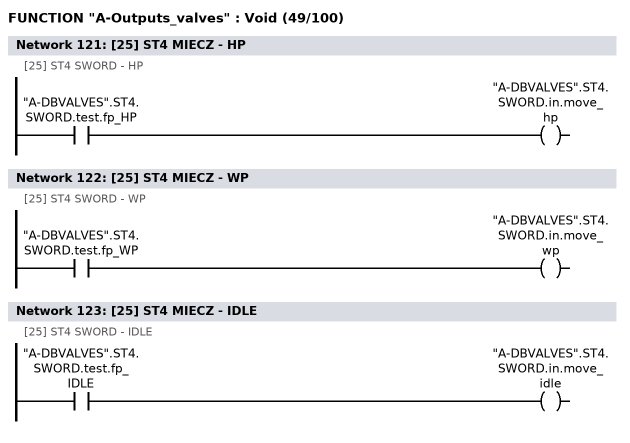
      O "A-DBVALVES".ST4.SWORD.test.fp_HP;
//    O     "A-Flags".STATION.IN_HP_STEP
      = "A-DBVALVES".ST4.SWORD.in.move_hp;
NETWORK
TITLE = [25] ST4 MIECZ - WP
//[25] ST4 SWORD - WP
      O "A-DBVALVES".ST4.SWORD.test.fp_WP;
      = "A-DBVALVES".ST4.SWORD.in.move_wp;
NETWORK
TITLE = [25] ST4 MIECZ - IDLE
//[25] ST4 SWORD - IDLE
      O "A-DBVALVES".ST4.SWORD.test.fp_IDLE;
      = "A-DBVALVES".ST4.SWORD.in.move_idle;
NETWORK
TITLE = [25] ST4 MIECZ
//[25] ST4 SWORD
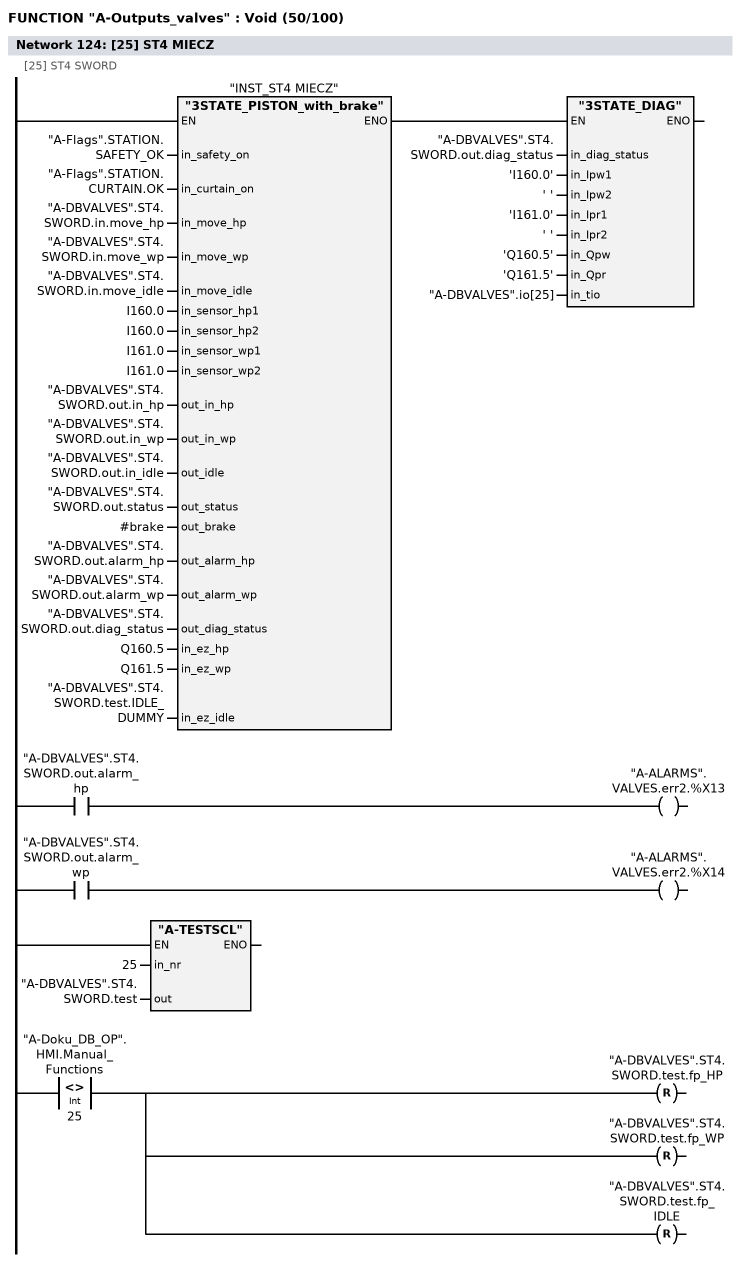
      CALL "3STATE_PISTON_with_brake", "INST_ST4 MIECZ"
      (  in_safety_on                := "A-Flags".STATION.SAFETY_OK ,
         in_curtain_on               := "A-Flags".STATION.CURTAIN.OK ,
         in_move_hp                  := "A-DBVALVES".ST4.SWORD.in.move_hp ,
         in_move_wp                  := "A-DBVALVES".ST4.SWORD.in.move_wp ,
         in_move_idle                := "A-DBVALVES".ST4.SWORD.in.move_idle ,
         in_sensor_hp1               := I160.0 ,
         in_sensor_hp2               := I160.0 ,
         in_sensor_wp1               := I161.0 ,
         in_sensor_wp2               := I161.0 ,
         out_in_hp                   := "A-DBVALVES".ST4.SWORD.out.in_hp ,
         out_in_wp                   := "A-DBVALVES".ST4.SWORD.out.in_wp ,
         out_idle                    := "A-DBVALVES".ST4.SWORD.out.in_idle ,
         out_status                  := "A-DBVALVES".ST4.SWORD.out.status ,
         out_brake                   := #brake ,
         out_alarm_hp                := "A-DBVALVES".ST4.SWORD.out.alarm_hp ,
         out_alarm_wp                := "A-DBVALVES".ST4.SWORD.out.alarm_wp ,
         out_diag_status             := "A-DBVALVES".ST4.SWORD.out.diag_status ,
         in_ez_hp                    := Q160.5 ,
         in_ez_wp                    := Q161.5 ,
         in_ez_idle                  := "A-DBVALVES".ST4.SWORD.test.IDLE_DUMMY
      );

      CALL "3STATE_DIAG"
      (  in_diag_status              := "A-DBVALVES".ST4.SWORD.out.diag_status ,
         in_Ipw1                     := 'I160.0' ,
         in_Ipw2                     := ' ' ,
         in_Ipr1                     := 'I161.0' ,
         in_Ipr2                     := ' ' ,
         in_Qpw                      := 'Q160.5' ,
         in_Qpr                      := 'Q161.5' ,
         in_tio                      := "A-DBVALVES".io[25]
      );

      A "A-DBVALVES".ST4.SWORD.out.alarm_hp;
      = "A-ALARMS".VALVES.err2.%X13;

      A "A-DBVALVES".ST4.SWORD.out.alarm_wp;
      = "A-ALARMS".VALVES.err2.%X14;

      CALL "A-TESTSCL"
      (  in_nr                       := 25 ,
         out                         := "A-DBVALVES".ST4.SWORD.test
      );

      A(;
      L "A-Doku_DB_OP".HMI.Manual_Functions;
      L 25;
      <>I;
      );
      R "A-DBVALVES".ST4.SWORD.test.fp_HP;
      R "A-DBVALVES".ST4.SWORD.test.fp_WP;
      R "A-DBVALVES".ST4.SWORD.test.fp_IDLE;
NETWORK
TITLE = -

NETWORK
TITLE = [26] ST4 ZDERZAK - HP
//[26] ST4 BUMPER - HP
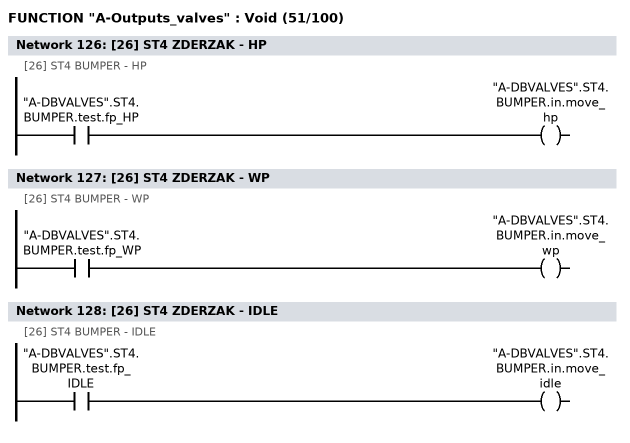
      O "A-DBVALVES".ST4.BUMPER.test.fp_HP;
//    O     "A-Flags".STATION.IN_HP_STEP
      = "A-DBVALVES".ST4.BUMPER.in.move_hp;
NETWORK
TITLE = [26] ST4 ZDERZAK - WP
//[26] ST4 BUMPER - WP
      O "A-DBVALVES".ST4.BUMPER.test.fp_WP;
      = "A-DBVALVES".ST4.BUMPER.in.move_wp;
NETWORK
TITLE = [26] ST4 ZDERZAK - IDLE
//[26] ST4 BUMPER - IDLE
      O "A-DBVALVES".ST4.BUMPER.test.fp_IDLE;
      = "A-DBVALVES".ST4.BUMPER.in.move_idle;
NETWORK
TITLE = [26] ST4 ZDERZAK
//[26] ST4 BUMPER
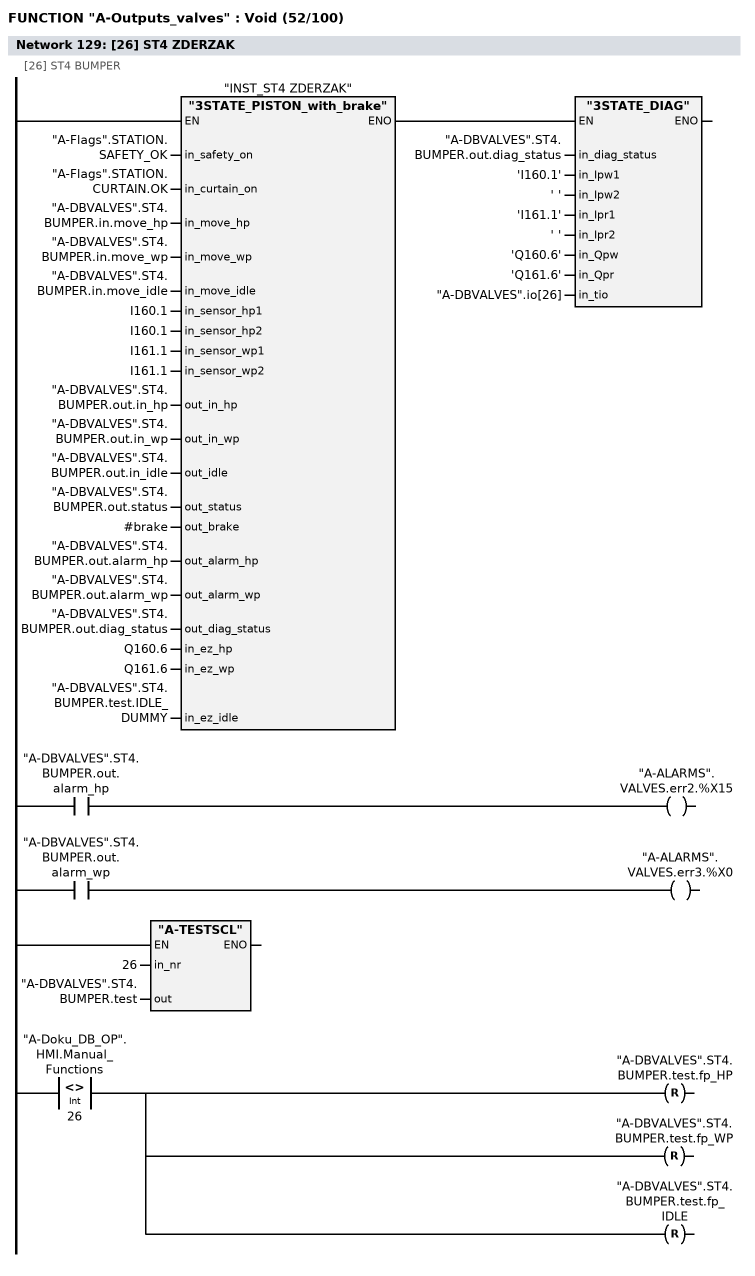
      CALL "3STATE_PISTON_with_brake", "INST_ST4 ZDERZAK"
      (  in_safety_on                := "A-Flags".STATION.SAFETY_OK ,
         in_curtain_on               := "A-Flags".STATION.CURTAIN.OK ,
         in_move_hp                  := "A-DBVALVES".ST4.BUMPER.in.move_hp ,
         in_move_wp                  := "A-DBVALVES".ST4.BUMPER.in.move_wp ,
         in_move_idle                := "A-DBVALVES".ST4.BUMPER.in.move_idle ,
         in_sensor_hp1               := I160.1 ,
         in_sensor_hp2               := I160.1 ,
         in_sensor_wp1               := I161.1 ,
         in_sensor_wp2               := I161.1 ,
         out_in_hp                   := "A-DBVALVES".ST4.BUMPER.out.in_hp ,
         out_in_wp                   := "A-DBVALVES".ST4.BUMPER.out.in_wp ,
         out_idle                    := "A-DBVALVES".ST4.BUMPER.out.in_idle ,
         out_status                  := "A-DBVALVES".ST4.BUMPER.out.status ,
         out_brake                   := #brake ,
         out_alarm_hp                := "A-DBVALVES".ST4.BUMPER.out.alarm_hp ,
         out_alarm_wp                := "A-DBVALVES".ST4.BUMPER.out.alarm_wp ,
         out_diag_status             := "A-DBVALVES".ST4.BUMPER.out.diag_status ,
         in_ez_hp                    := Q160.6 ,
         in_ez_wp                    := Q161.6 ,
         in_ez_idle                  := "A-DBVALVES".ST4.BUMPER.test.IDLE_DUMMY
      );

      CALL "3STATE_DIAG"
      (  in_diag_status              := "A-DBVALVES".ST4.BUMPER.out.diag_status ,
         in_Ipw1                     := 'I160.1' ,
         in_Ipw2                     := ' ' ,
         in_Ipr1                     := 'I161.1' ,
         in_Ipr2                     := ' ' ,
         in_Qpw                      := 'Q160.6' ,
         in_Qpr                      := 'Q161.6' ,
         in_tio                      := "A-DBVALVES".io[26]
      );

      A "A-DBVALVES".ST4.BUMPER.out.alarm_hp;
      = "A-ALARMS".VALVES.err2.%X15;

      A "A-DBVALVES".ST4.BUMPER.out.alarm_wp;
      = "A-ALARMS".VALVES.err3.%X0;

      CALL "A-TESTSCL"
      (  in_nr                       := 26 ,
         out                         := "A-DBVALVES".ST4.BUMPER.test
      );

      A(;
      L "A-Doku_DB_OP".HMI.Manual_Functions;
      L 26;
      <>I;
      );
      R "A-DBVALVES".ST4.BUMPER.test.fp_HP;
      R "A-DBVALVES".ST4.BUMPER.test.fp_WP;
      R "A-DBVALVES".ST4.BUMPER.test.fp_IDLE;
NETWORK
TITLE = -

NETWORK
TITLE = [27] ST4 PODNOSZENIE_MIECZA - HP
//[27] ST4 SWORD_RISING - HP
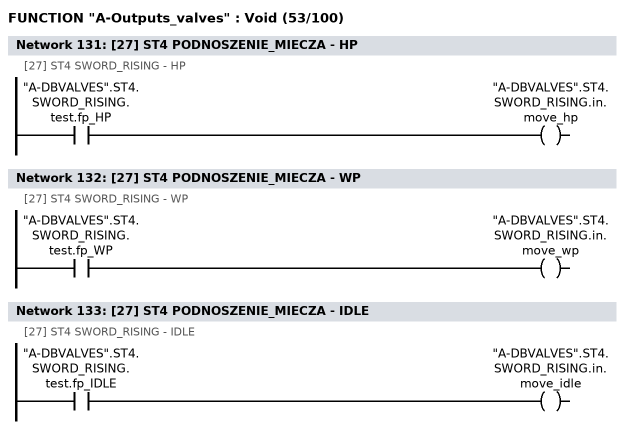
      O "A-DBVALVES".ST4.SWORD_RISING.test.fp_HP;
//    O     "A-Flags".STATION.IN_HP_STEP
      = "A-DBVALVES".ST4.SWORD_RISING.in.move_hp;
NETWORK
TITLE = [27] ST4 PODNOSZENIE_MIECZA - WP
//[27] ST4 SWORD_RISING - WP
      O "A-DBVALVES".ST4.SWORD_RISING.test.fp_WP;
      = "A-DBVALVES".ST4.SWORD_RISING.in.move_wp;
NETWORK
TITLE = [27] ST4 PODNOSZENIE_MIECZA - IDLE
//[27] ST4 SWORD_RISING - IDLE
      O "A-DBVALVES".ST4.SWORD_RISING.test.fp_IDLE;
      = "A-DBVALVES".ST4.SWORD_RISING.in.move_idle;
NETWORK
TITLE = [27] ST4 PODNOSZENIE_MIECZA
//[27] ST4 SWORD_RISING
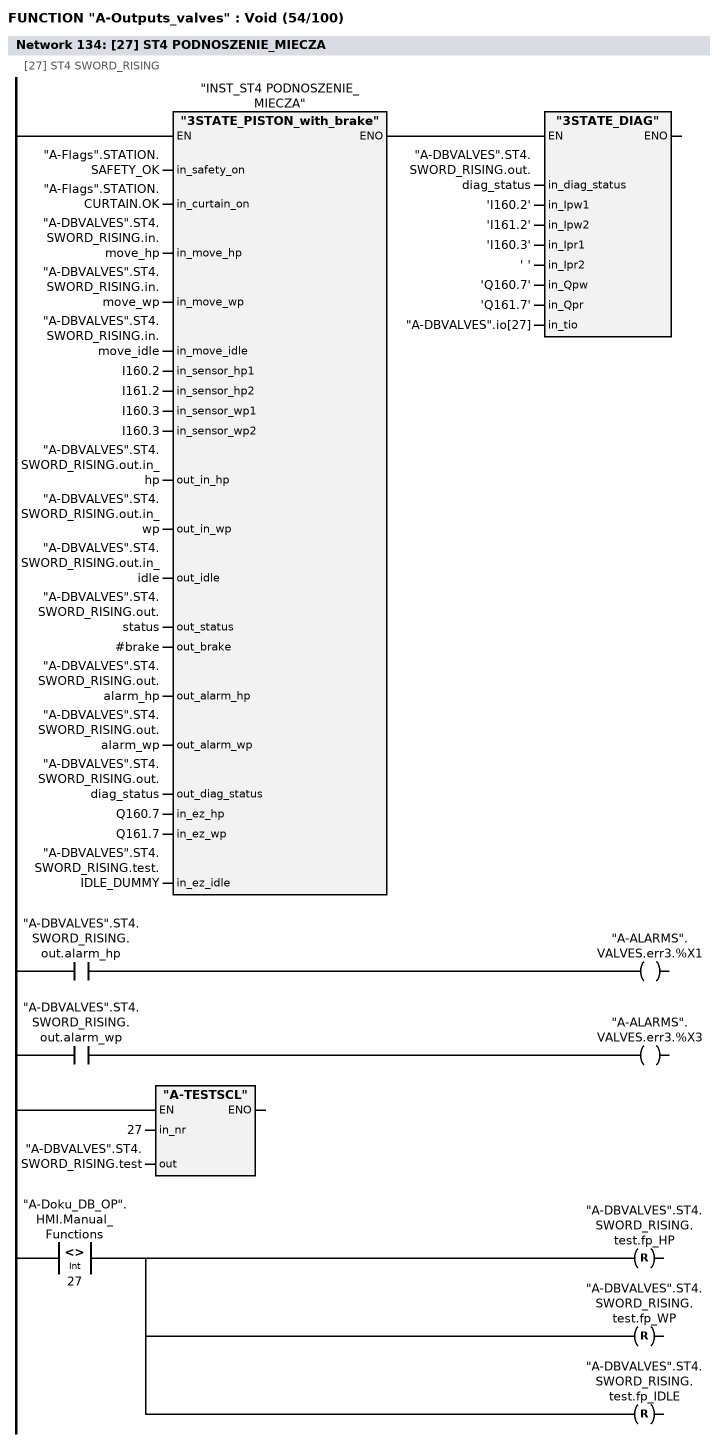
      CALL "3STATE_PISTON_with_brake", "INST_ST4 PODNOSZENIE_MIECZA"
      (  in_safety_on                := "A-Flags".STATION.SAFETY_OK ,
         in_curtain_on               := "A-Flags".STATION.CURTAIN.OK ,
         in_move_hp                  := "A-DBVALVES".ST4.SWORD_RISING.in.move_hp ,
         in_move_wp                  := "A-DBVALVES".ST4.SWORD_RISING.in.move_wp ,
         in_move_idle                := "A-DBVALVES".ST4.SWORD_RISING.in.move_idle ,
         in_sensor_hp1               := I160.2 ,
         in_sensor_hp2               := I161.2 ,
         in_sensor_wp1               := I160.3 ,
         in_sensor_wp2               := I160.3 ,
         out_in_hp                   := "A-DBVALVES".ST4.SWORD_RISING.out.in_hp ,
         out_in_wp                   := "A-DBVALVES".ST4.SWORD_RISING.out.in_wp ,
         out_idle                    := "A-DBVALVES".ST4.SWORD_RISING.out.in_idle ,
         out_status                  := "A-DBVALVES".ST4.SWORD_RISING.out.status ,
         out_brake                   := #brake ,
         out_alarm_hp                := "A-DBVALVES".ST4.SWORD_RISING.out.alarm_hp ,
         out_alarm_wp                := "A-DBVALVES".ST4.SWORD_RISING.out.alarm_wp ,
         out_diag_status             := "A-DBVALVES".ST4.SWORD_RISING.out.diag_status ,
         in_ez_hp                    := Q160.7 ,
         in_ez_wp                    := Q161.7 ,
         in_ez_idle                  := "A-DBVALVES".ST4.SWORD_RISING.test.IDLE_DUMMY
      );

      CALL "3STATE_DIAG"
      (  in_diag_status              := "A-DBVALVES".ST4.SWORD_RISING.out.diag_status ,
         in_Ipw1                     := 'I160.2' ,
         in_Ipw2                     := 'I161.2' ,
         in_Ipr1                     := 'I160.3' ,
         in_Ipr2                     := ' ' ,
         in_Qpw                      := 'Q160.7' ,
         in_Qpr                      := 'Q161.7' ,
         in_tio                      := "A-DBVALVES".io[27]
      );

      A "A-DBVALVES".ST4.SWORD_RISING.out.alarm_hp;
      = "A-ALARMS".VALVES.err3.%X1;

      A "A-DBVALVES".ST4.SWORD_RISING.out.alarm_wp;
      = "A-ALARMS".VALVES.err3.%X3;

      CALL "A-TESTSCL"
      (  in_nr                       := 27 ,
         out                         := "A-DBVALVES".ST4.SWORD_RISING.test
      );

      A(;
      L "A-Doku_DB_OP".HMI.Manual_Functions;
      L 27;
      <>I;
      );
      R "A-DBVALVES".ST4.SWORD_RISING.test.fp_HP;
      R "A-DBVALVES".ST4.SWORD_RISING.test.fp_WP;
      R "A-DBVALVES".ST4.SWORD_RISING.test.fp_IDLE;
NETWORK
TITLE = -

NETWORK
TITLE = [28] ST5 PRZESUW_STACJI - HP
//[28] ST5 STATION_MOVEMENT - HP
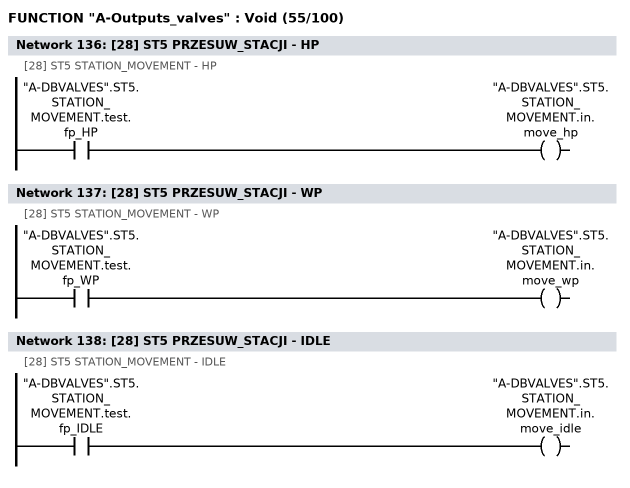
      O "A-DBVALVES".ST5.STATION_MOVEMENT.test.fp_HP;
//    O     "A-Flags".STATION.IN_HP_STEP
      = "A-DBVALVES".ST5.STATION_MOVEMENT.in.move_hp;
NETWORK
TITLE = [28] ST5 PRZESUW_STACJI - WP
//[28] ST5 STATION_MOVEMENT - WP
      O "A-DBVALVES".ST5.STATION_MOVEMENT.test.fp_WP;
      = "A-DBVALVES".ST5.STATION_MOVEMENT.in.move_wp;
NETWORK
TITLE = [28] ST5 PRZESUW_STACJI - IDLE
//[28] ST5 STATION_MOVEMENT - IDLE
      O "A-DBVALVES".ST5.STATION_MOVEMENT.test.fp_IDLE;
      = "A-DBVALVES".ST5.STATION_MOVEMENT.in.move_idle;
NETWORK
TITLE = [28] ST5 PRZESUW_STACJI
//[28] ST5 STATION_MOVEMENT
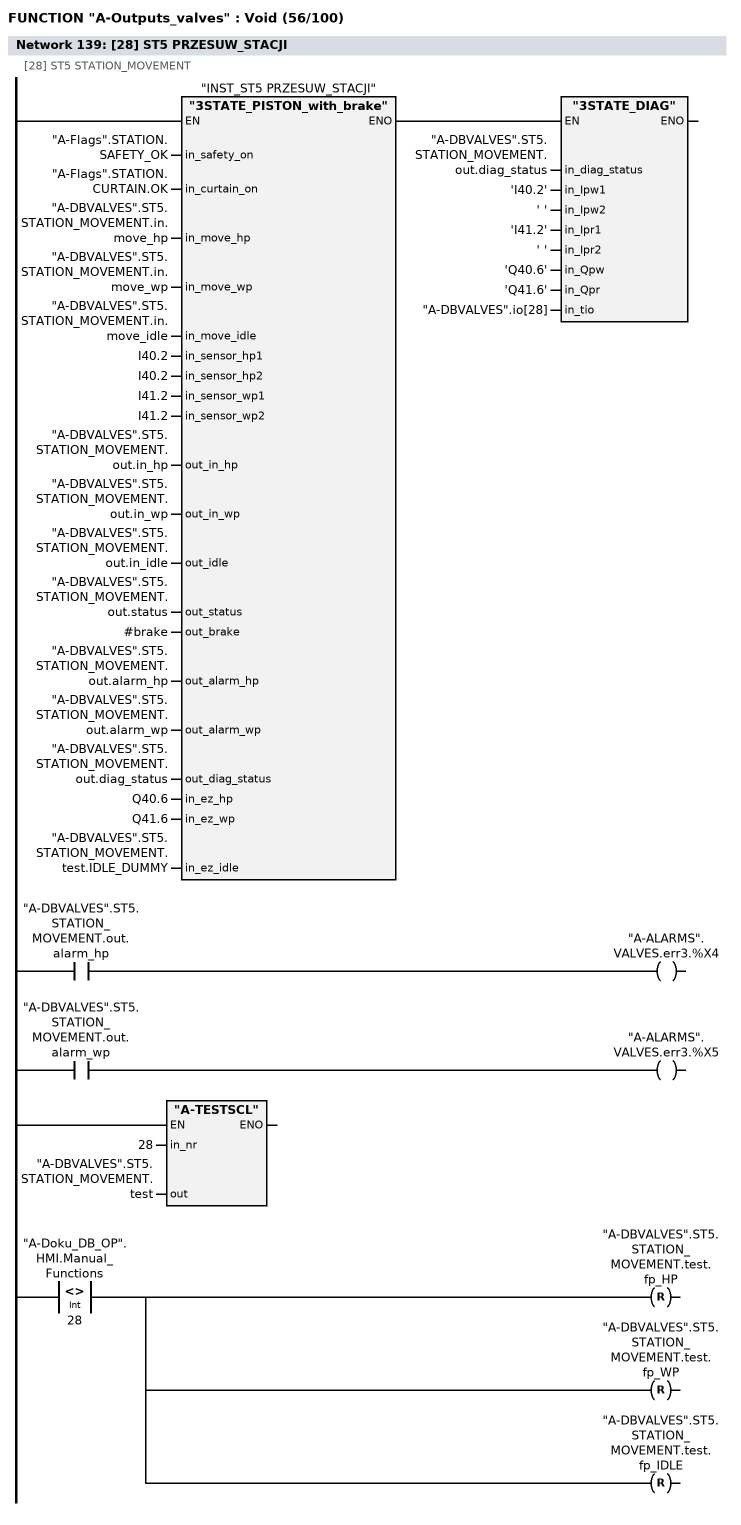
      CALL "3STATE_PISTON_with_brake", "INST_ST5 PRZESUW_STACJI"
      (  in_safety_on                := "A-Flags".STATION.SAFETY_OK ,
         in_curtain_on               := "A-Flags".STATION.CURTAIN.OK ,
         in_move_hp                  := "A-DBVALVES".ST5.STATION_MOVEMENT.in.move_hp ,
         in_move_wp                  := "A-DBVALVES".ST5.STATION_MOVEMENT.in.move_wp ,
         in_move_idle                := "A-DBVALVES".ST5.STATION_MOVEMENT.in.move_idle ,
         in_sensor_hp1               := I40.2 ,
         in_sensor_hp2               := I40.2 ,
         in_sensor_wp1               := I41.2 ,
         in_sensor_wp2               := I41.2 ,
         out_in_hp                   := "A-DBVALVES".ST5.STATION_MOVEMENT.out.in_hp ,
         out_in_wp                   := "A-DBVALVES".ST5.STATION_MOVEMENT.out.in_wp ,
         out_idle                    := "A-DBVALVES".ST5.STATION_MOVEMENT.out.in_idle ,
         out_status                  := "A-DBVALVES".ST5.STATION_MOVEMENT.out.status ,
         out_brake                   := #brake ,
         out_alarm_hp                := "A-DBVALVES".ST5.STATION_MOVEMENT.out.alarm_hp ,
         out_alarm_wp                := "A-DBVALVES".ST5.STATION_MOVEMENT.out.alarm_wp ,
         out_diag_status             := "A-DBVALVES".ST5.STATION_MOVEMENT.out.diag_status ,
         in_ez_hp                    := Q40.6 ,
         in_ez_wp                    := Q41.6 ,
         in_ez_idle                  := "A-DBVALVES".ST5.STATION_MOVEMENT.test.IDLE_DUMMY
      );

      CALL "3STATE_DIAG"
      (  in_diag_status              := "A-DBVALVES".ST5.STATION_MOVEMENT.out.diag_status ,
         in_Ipw1                     := 'I40.2' ,
         in_Ipw2                     := ' ' ,
         in_Ipr1                     := 'I41.2' ,
         in_Ipr2                     := ' ' ,
         in_Qpw                      := 'Q40.6' ,
         in_Qpr                      := 'Q41.6' ,
         in_tio                      := "A-DBVALVES".io[28]
      );

      A "A-DBVALVES".ST5.STATION_MOVEMENT.out.alarm_hp;
      = "A-ALARMS".VALVES.err3.%X4;

      A "A-DBVALVES".ST5.STATION_MOVEMENT.out.alarm_wp;
      = "A-ALARMS".VALVES.err3.%X5;

      CALL "A-TESTSCL"
      (  in_nr                       := 28 ,
         out                         := "A-DBVALVES".ST5.STATION_MOVEMENT.test
      );

      A(;
      L "A-Doku_DB_OP".HMI.Manual_Functions;
      L 28;
      <>I;
      );
      R "A-DBVALVES".ST5.STATION_MOVEMENT.test.fp_HP;
      R "A-DBVALVES".ST5.STATION_MOVEMENT.test.fp_WP;
      R "A-DBVALVES".ST5.STATION_MOVEMENT.test.fp_IDLE;
NETWORK
TITLE = -

NETWORK
TITLE = [29] ST5 STACJA_MALY_SKOK - HP
//[29] ST5 STATION_SMALL_STEP - HP
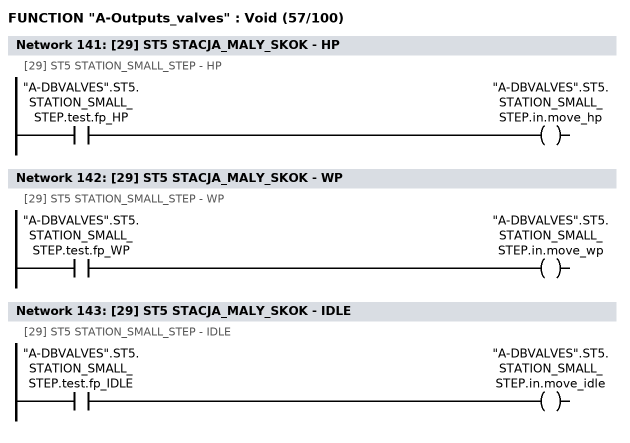
      O "A-DBVALVES".ST5.STATION_SMALL_STEP.test.fp_HP;
//    O     "A-Flags".STATION.IN_HP_STEP
      = "A-DBVALVES".ST5.STATION_SMALL_STEP.in.move_hp;
NETWORK
TITLE = [29] ST5 STACJA_MALY_SKOK - WP
//[29] ST5 STATION_SMALL_STEP - WP
      O "A-DBVALVES".ST5.STATION_SMALL_STEP.test.fp_WP;
      = "A-DBVALVES".ST5.STATION_SMALL_STEP.in.move_wp;
NETWORK
TITLE = [29] ST5 STACJA_MALY_SKOK - IDLE
//[29] ST5 STATION_SMALL_STEP - IDLE
      O "A-DBVALVES".ST5.STATION_SMALL_STEP.test.fp_IDLE;
      = "A-DBVALVES".ST5.STATION_SMALL_STEP.in.move_idle;
NETWORK
TITLE = [29] ST5 STACJA_MALY_SKOK
//[29] ST5 STATION_SMALL_STEP
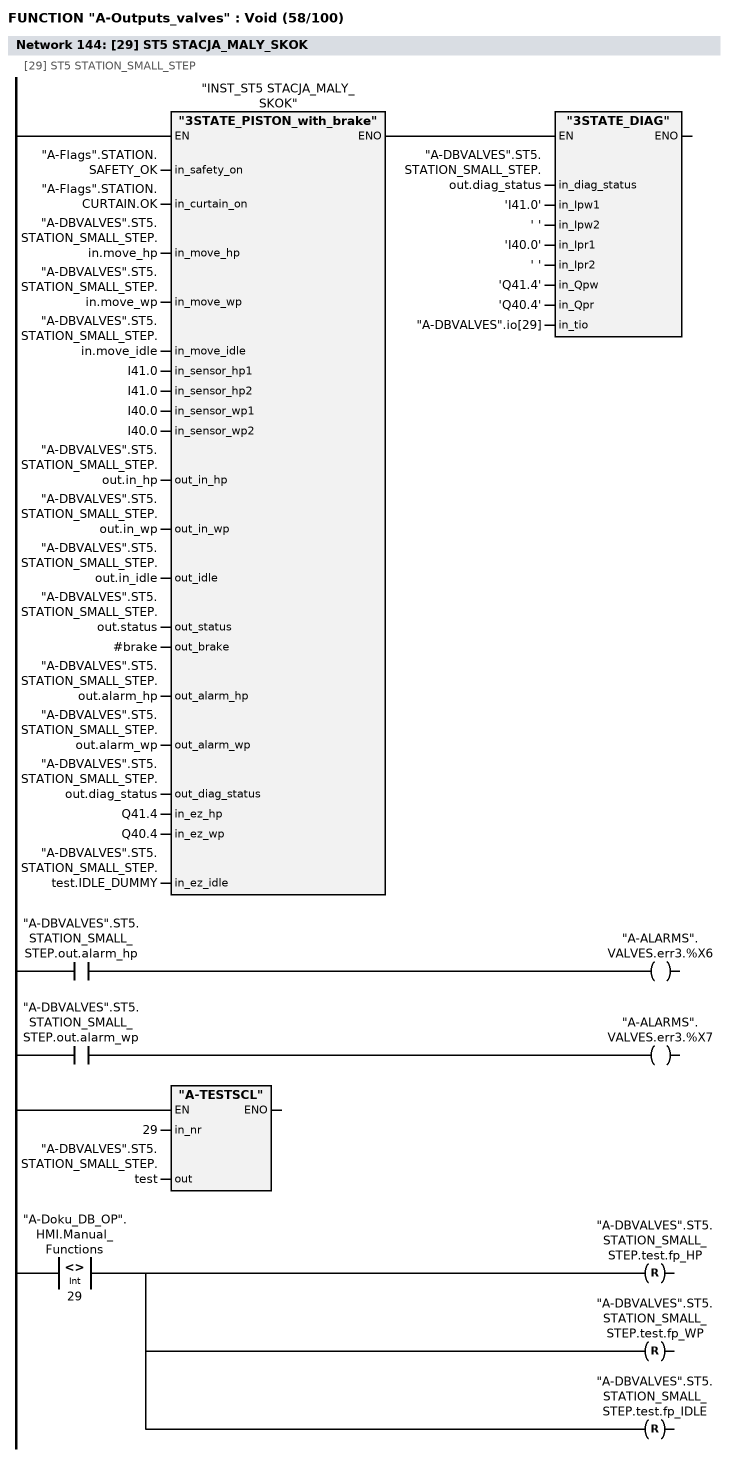
      CALL "3STATE_PISTON_with_brake", "INST_ST5 STACJA_MALY_SKOK"
      (  in_safety_on                := "A-Flags".STATION.SAFETY_OK ,
         in_curtain_on               := "A-Flags".STATION.CURTAIN.OK ,
         in_move_hp                  := "A-DBVALVES".ST5.STATION_SMALL_STEP.in.move_hp ,
         in_move_wp                  := "A-DBVALVES".ST5.STATION_SMALL_STEP.in.move_wp ,
         in_move_idle                := "A-DBVALVES".ST5.STATION_SMALL_STEP.in.move_idle ,
         in_sensor_hp1               := I41.0 ,
         in_sensor_hp2               := I41.0 ,
         in_sensor_wp1               := I40.0 ,
         in_sensor_wp2               := I40.0 ,
         out_in_hp                   := "A-DBVALVES".ST5.STATION_SMALL_STEP.out.in_hp ,
         out_in_wp                   := "A-DBVALVES".ST5.STATION_SMALL_STEP.out.in_wp ,
         out_idle                    := "A-DBVALVES".ST5.STATION_SMALL_STEP.out.in_idle ,
         out_status                  := "A-DBVALVES".ST5.STATION_SMALL_STEP.out.status ,
         out_brake                   := #brake ,
         out_alarm_hp                := "A-DBVALVES".ST5.STATION_SMALL_STEP.out.alarm_hp ,
         out_alarm_wp                := "A-DBVALVES".ST5.STATION_SMALL_STEP.out.alarm_wp ,
         out_diag_status             := "A-DBVALVES".ST5.STATION_SMALL_STEP.out.diag_status ,
         in_ez_hp                    := Q41.4 ,
         in_ez_wp                    := Q40.4 ,
         in_ez_idle                  := "A-DBVALVES".ST5.STATION_SMALL_STEP.test.IDLE_DUMMY
      );

      CALL "3STATE_DIAG"
      (  in_diag_status              := "A-DBVALVES".ST5.STATION_SMALL_STEP.out.diag_status ,
         in_Ipw1                     := 'I41.0' ,
         in_Ipw2                     := ' ' ,
         in_Ipr1                     := 'I40.0' ,
         in_Ipr2                     := ' ' ,
         in_Qpw                      := 'Q41.4' ,
         in_Qpr                      := 'Q40.4' ,
         in_tio                      := "A-DBVALVES".io[29]
      );

      A "A-DBVALVES".ST5.STATION_SMALL_STEP.out.alarm_hp;
      = "A-ALARMS".VALVES.err3.%X6;

      A "A-DBVALVES".ST5.STATION_SMALL_STEP.out.alarm_wp;
      = "A-ALARMS".VALVES.err3.%X7;

      CALL "A-TESTSCL"
      (  in_nr                       := 29 ,
         out                         := "A-DBVALVES".ST5.STATION_SMALL_STEP.test
      );

      A(;
      L "A-Doku_DB_OP".HMI.Manual_Functions;
      L 29;
      <>I;
      );
      R "A-DBVALVES".ST5.STATION_SMALL_STEP.test.fp_HP;
      R "A-DBVALVES".ST5.STATION_SMALL_STEP.test.fp_WP;
      R "A-DBVALVES".ST5.STATION_SMALL_STEP.test.fp_IDLE;
NETWORK
TITLE = -

NETWORK
TITLE = [30] ST5 STACJA_DUZY_SKOK - HP
//[30] ST5 STATION_BIG_STEP - HP
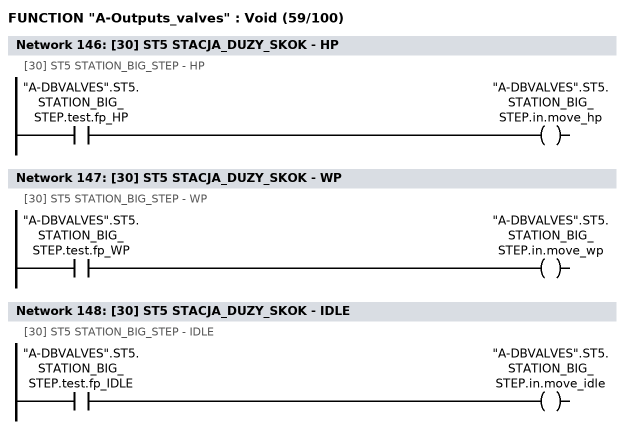
      O "A-DBVALVES".ST5.STATION_BIG_STEP.test.fp_HP;
//    O     "A-Flags".STATION.IN_HP_STEP
      = "A-DBVALVES".ST5.STATION_BIG_STEP.in.move_hp;
NETWORK
TITLE = [30] ST5 STACJA_DUZY_SKOK - WP
//[30] ST5 STATION_BIG_STEP - WP
      O "A-DBVALVES".ST5.STATION_BIG_STEP.test.fp_WP;
      = "A-DBVALVES".ST5.STATION_BIG_STEP.in.move_wp;
NETWORK
TITLE = [30] ST5 STACJA_DUZY_SKOK - IDLE
//[30] ST5 STATION_BIG_STEP - IDLE
      O "A-DBVALVES".ST5.STATION_BIG_STEP.test.fp_IDLE;
      = "A-DBVALVES".ST5.STATION_BIG_STEP.in.move_idle;
NETWORK
TITLE = [30] ST5 STACJA_DUZY_SKOK
//[30] ST5 STATION_BIG_STEP
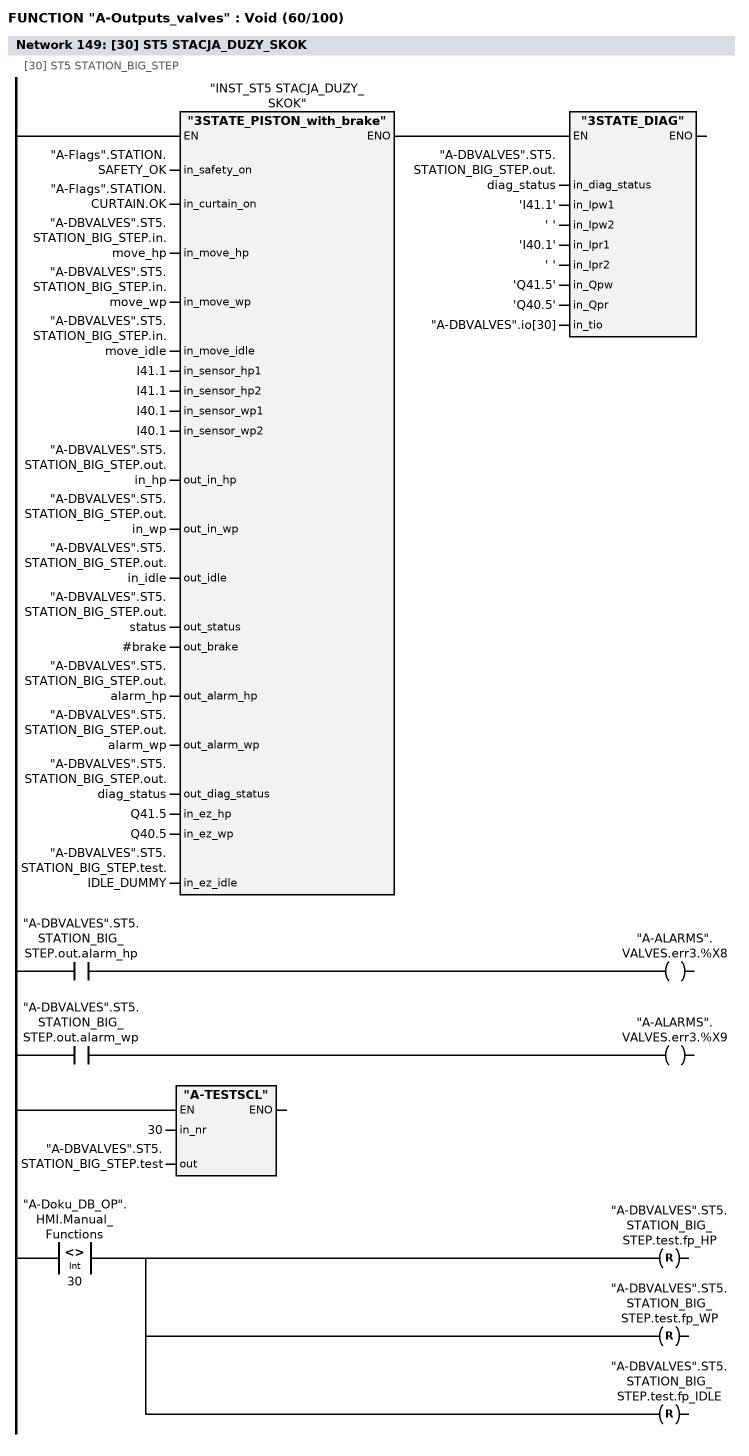
      CALL "3STATE_PISTON_with_brake", "INST_ST5 STACJA_DUZY_SKOK"
      (  in_safety_on                := "A-Flags".STATION.SAFETY_OK ,
         in_curtain_on               := "A-Flags".STATION.CURTAIN.OK ,
         in_move_hp                  := "A-DBVALVES".ST5.STATION_BIG_STEP.in.move_hp ,
         in_move_wp                  := "A-DBVALVES".ST5.STATION_BIG_STEP.in.move_wp ,
         in_move_idle                := "A-DBVALVES".ST5.STATION_BIG_STEP.in.move_idle ,
         in_sensor_hp1               := I41.1 ,
         in_sensor_hp2               := I41.1 ,
         in_sensor_wp1               := I40.1 ,
         in_sensor_wp2               := I40.1 ,
         out_in_hp                   := "A-DBVALVES".ST5.STATION_BIG_STEP.out.in_hp ,
         out_in_wp                   := "A-DBVALVES".ST5.STATION_BIG_STEP.out.in_wp ,
         out_idle                    := "A-DBVALVES".ST5.STATION_BIG_STEP.out.in_idle ,
         out_status                  := "A-DBVALVES".ST5.STATION_BIG_STEP.out.status ,
         out_brake                   := #brake ,
         out_alarm_hp                := "A-DBVALVES".ST5.STATION_BIG_STEP.out.alarm_hp ,
         out_alarm_wp                := "A-DBVALVES".ST5.STATION_BIG_STEP.out.alarm_wp ,
         out_diag_status             := "A-DBVALVES".ST5.STATION_BIG_STEP.out.diag_status ,
         in_ez_hp                    := Q41.5 ,
         in_ez_wp                    := Q40.5 ,
         in_ez_idle                  := "A-DBVALVES".ST5.STATION_BIG_STEP.test.IDLE_DUMMY
      );

      CALL "3STATE_DIAG"
      (  in_diag_status              := "A-DBVALVES".ST5.STATION_BIG_STEP.out.diag_status ,
         in_Ipw1                     := 'I41.1' ,
         in_Ipw2                     := ' ' ,
         in_Ipr1                     := 'I40.1' ,
         in_Ipr2                     := ' ' ,
         in_Qpw                      := 'Q41.5' ,
         in_Qpr                      := 'Q40.5' ,
         in_tio                      := "A-DBVALVES".io[30]
      );

      A "A-DBVALVES".ST5.STATION_BIG_STEP.out.alarm_hp;
      = "A-ALARMS".VALVES.err3.%X8;

      A "A-DBVALVES".ST5.STATION_BIG_STEP.out.alarm_wp;
      = "A-ALARMS".VALVES.err3.%X9;

      CALL "A-TESTSCL"
      (  in_nr                       := 30 ,
         out                         := "A-DBVALVES".ST5.STATION_BIG_STEP.test
      );

      A(;
      L "A-Doku_DB_OP".HMI.Manual_Functions;
      L 30;
      <>I;
      );
      R "A-DBVALVES".ST5.STATION_BIG_STEP.test.fp_HP;
      R "A-DBVALVES".ST5.STATION_BIG_STEP.test.fp_WP;
      R "A-DBVALVES".ST5.STATION_BIG_STEP.test.fp_IDLE;
NETWORK
TITLE = -

NETWORK
TITLE = [31] ST5 PIN - HP
//[31] ST5 PIN - HP
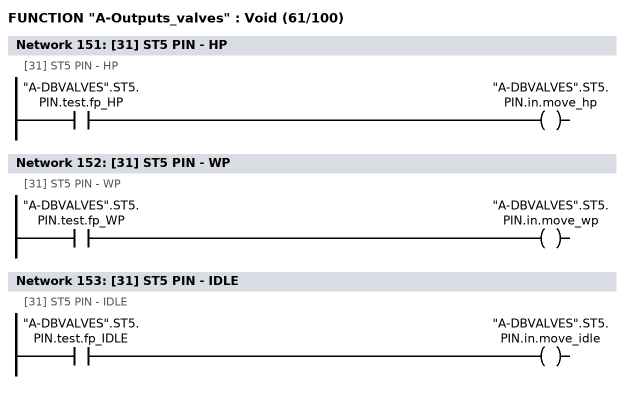
      O "A-DBVALVES".ST5.PIN.test.fp_HP;
//    O     "A-Flags".STATION.IN_HP_STEP
      = "A-DBVALVES".ST5.PIN.in.move_hp;
NETWORK
TITLE = [31] ST5 PIN - WP
//[31] ST5 PIN - WP
      O "A-DBVALVES".ST5.PIN.test.fp_WP;
      = "A-DBVALVES".ST5.PIN.in.move_wp;
NETWORK
TITLE = [31] ST5 PIN - IDLE
//[31] ST5 PIN - IDLE
      O "A-DBVALVES".ST5.PIN.test.fp_IDLE;
      = "A-DBVALVES".ST5.PIN.in.move_idle;
NETWORK
TITLE = [31] ST5 PIN
//[31] ST5 PIN
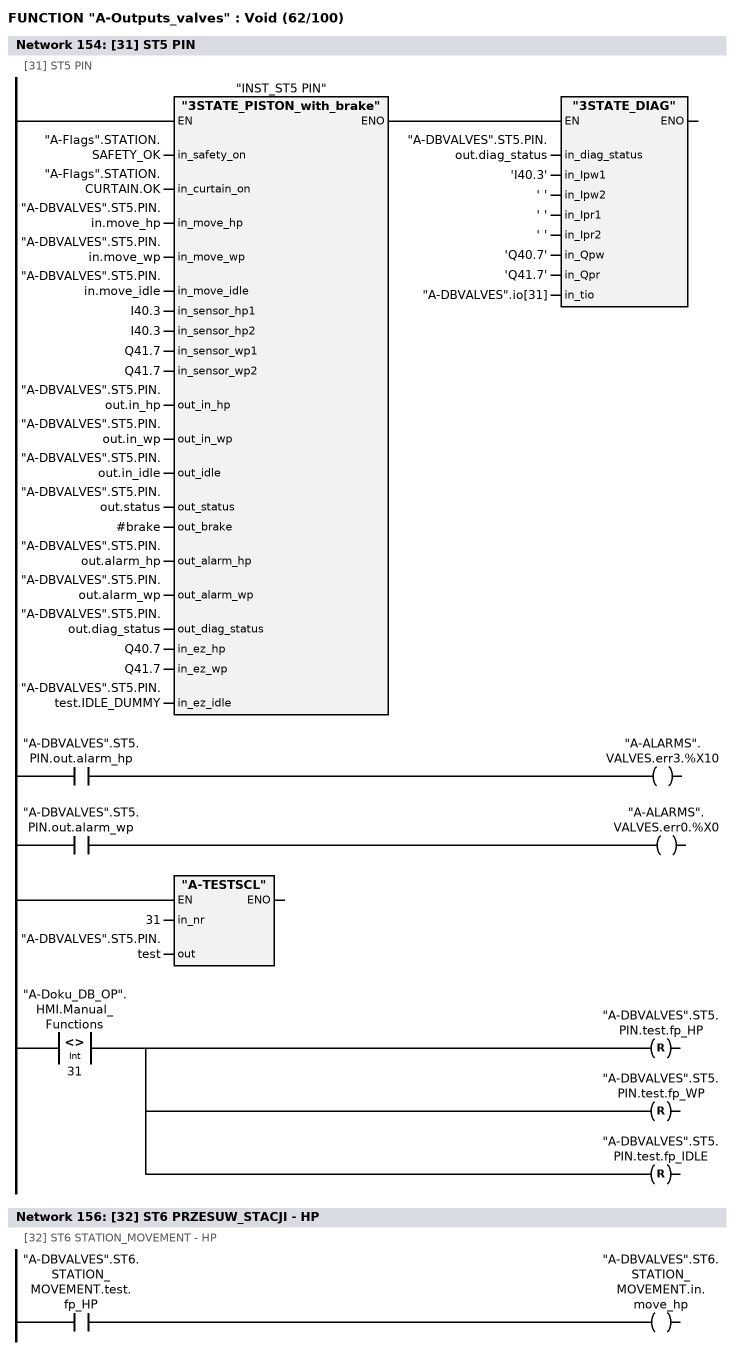
      CALL "3STATE_PISTON_with_brake", "INST_ST5 PIN"
      (  in_safety_on                := "A-Flags".STATION.SAFETY_OK ,
         in_curtain_on               := "A-Flags".STATION.CURTAIN.OK ,
         in_move_hp                  := "A-DBVALVES".ST5.PIN.in.move_hp ,
         in_move_wp                  := "A-DBVALVES".ST5.PIN.in.move_wp ,
         in_move_idle                := "A-DBVALVES".ST5.PIN.in.move_idle ,
         in_sensor_hp1               := I40.3 ,
         in_sensor_hp2               := I40.3 ,
         in_sensor_wp1               := Q41.7 ,
         in_sensor_wp2               := Q41.7 ,
         out_in_hp                   := "A-DBVALVES".ST5.PIN.out.in_hp ,
         out_in_wp                   := "A-DBVALVES".ST5.PIN.out.in_wp ,
         out_idle                    := "A-DBVALVES".ST5.PIN.out.in_idle ,
         out_status                  := "A-DBVALVES".ST5.PIN.out.status ,
         out_brake                   := #brake ,
         out_alarm_hp                := "A-DBVALVES".ST5.PIN.out.alarm_hp ,
         out_alarm_wp                := "A-DBVALVES".ST5.PIN.out.alarm_wp ,
         out_diag_status             := "A-DBVALVES".ST5.PIN.out.diag_status ,
         in_ez_hp                    := Q40.7 ,
         in_ez_wp                    := Q41.7 ,
         in_ez_idle                  := "A-DBVALVES".ST5.PIN.test.IDLE_DUMMY
      );

      CALL "3STATE_DIAG"
      (  in_diag_status              := "A-DBVALVES".ST5.PIN.out.diag_status ,
         in_Ipw1                     := 'I40.3' ,
         in_Ipw2                     := ' ' ,
         in_Ipr1                     := ' ' ,
         in_Ipr2                     := ' ' ,
         in_Qpw                      := 'Q40.7' ,
         in_Qpr                      := 'Q41.7' ,
         in_tio                      := "A-DBVALVES".io[31]
      );

      A "A-DBVALVES".ST5.PIN.out.alarm_hp;
      = "A-ALARMS".VALVES.err3.%X10;

      A "A-DBVALVES".ST5.PIN.out.alarm_wp;
      = "A-ALARMS".VALVES.err0.%X0;

      CALL "A-TESTSCL"
      (  in_nr                       := 31 ,
         out                         := "A-DBVALVES".ST5.PIN.test
      );

      A(;
      L "A-Doku_DB_OP".HMI.Manual_Functions;
      L 31;
      <>I;
      );
      R "A-DBVALVES".ST5.PIN.test.fp_HP;
      R "A-DBVALVES".ST5.PIN.test.fp_WP;
      R "A-DBVALVES".ST5.PIN.test.fp_IDLE;
NETWORK
TITLE = -

NETWORK
TITLE = [32] ST6 PRZESUW_STACJI - HP
//[32] ST6 STATION_MOVEMENT - HP
      O "A-DBVALVES".ST6.STATION_MOVEMENT.test.fp_HP;
//    O     "A-Flags".STATION.IN_HP_STEP
      = "A-DBVALVES".ST6.STATION_MOVEMENT.in.move_hp;
NETWORK
TITLE = [32] ST6 PRZESUW_STACJI - WP
//[32] ST6 STATION_MOVEMENT - WP
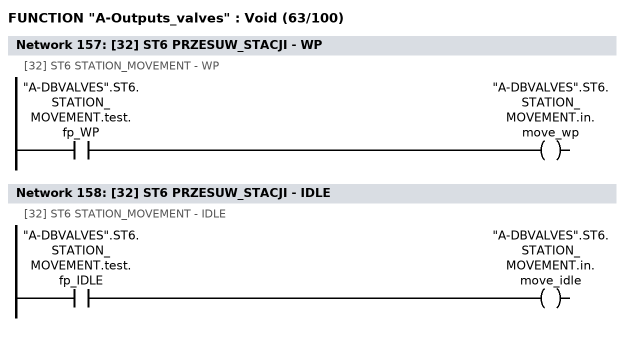
      O "A-DBVALVES".ST6.STATION_MOVEMENT.test.fp_WP;
      = "A-DBVALVES".ST6.STATION_MOVEMENT.in.move_wp;
NETWORK
TITLE = [32] ST6 PRZESUW_STACJI - IDLE
//[32] ST6 STATION_MOVEMENT - IDLE
      O "A-DBVALVES".ST6.STATION_MOVEMENT.test.fp_IDLE;
      = "A-DBVALVES".ST6.STATION_MOVEMENT.in.move_idle;
NETWORK
TITLE = [32] ST6 PRZESUW_STACJI
//[32] ST6 STATION_MOVEMENT
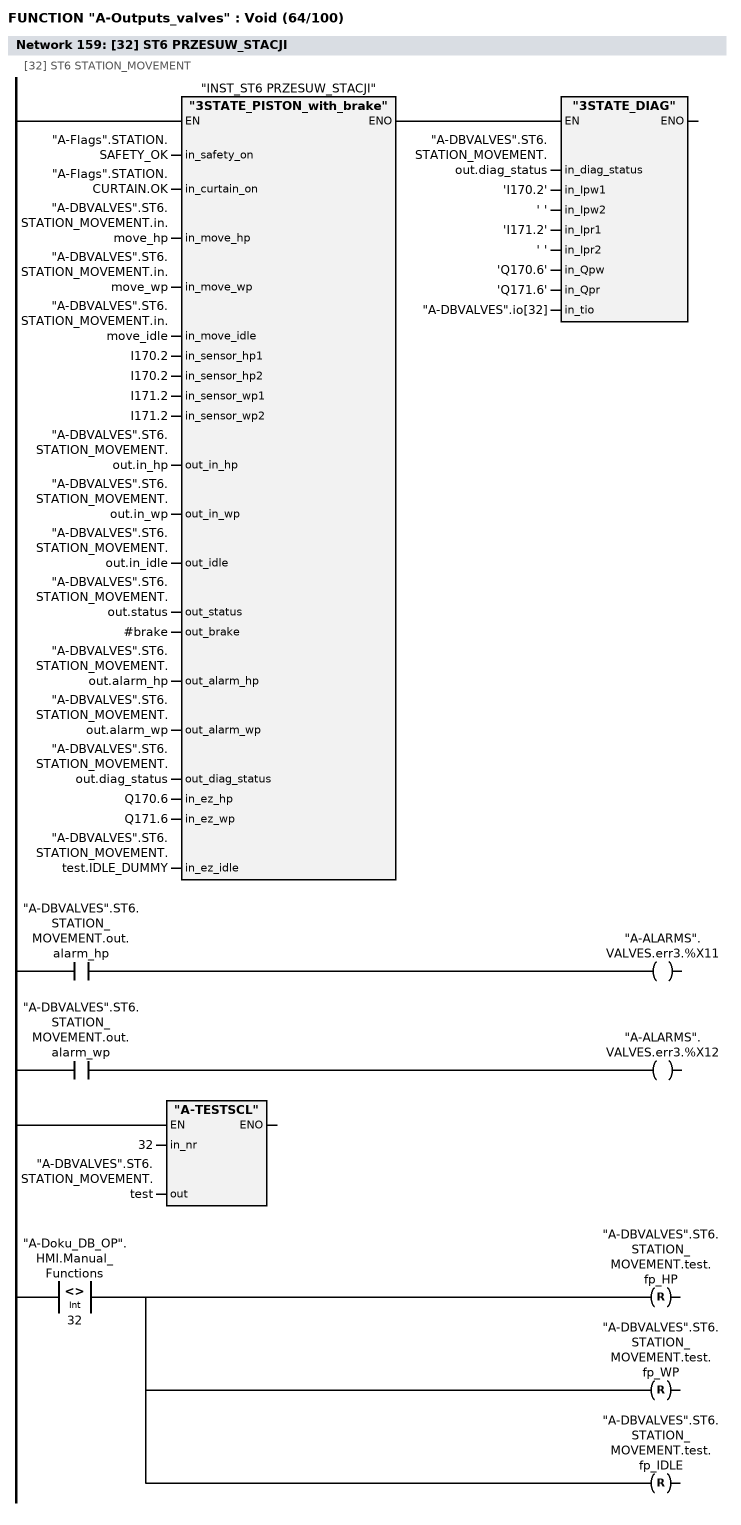
      CALL "3STATE_PISTON_with_brake", "INST_ST6 PRZESUW_STACJI"
      (  in_safety_on                := "A-Flags".STATION.SAFETY_OK ,
         in_curtain_on               := "A-Flags".STATION.CURTAIN.OK ,
         in_move_hp                  := "A-DBVALVES".ST6.STATION_MOVEMENT.in.move_hp ,
         in_move_wp                  := "A-DBVALVES".ST6.STATION_MOVEMENT.in.move_wp ,
         in_move_idle                := "A-DBVALVES".ST6.STATION_MOVEMENT.in.move_idle ,
         in_sensor_hp1               := I170.2 ,
         in_sensor_hp2               := I170.2 ,
         in_sensor_wp1               := I171.2 ,
         in_sensor_wp2               := I171.2 ,
         out_in_hp                   := "A-DBVALVES".ST6.STATION_MOVEMENT.out.in_hp ,
         out_in_wp                   := "A-DBVALVES".ST6.STATION_MOVEMENT.out.in_wp ,
         out_idle                    := "A-DBVALVES".ST6.STATION_MOVEMENT.out.in_idle ,
         out_status                  := "A-DBVALVES".ST6.STATION_MOVEMENT.out.status ,
         out_brake                   := #brake ,
         out_alarm_hp                := "A-DBVALVES".ST6.STATION_MOVEMENT.out.alarm_hp ,
         out_alarm_wp                := "A-DBVALVES".ST6.STATION_MOVEMENT.out.alarm_wp ,
         out_diag_status             := "A-DBVALVES".ST6.STATION_MOVEMENT.out.diag_status ,
         in_ez_hp                    := Q170.6 ,
         in_ez_wp                    := Q171.6 ,
         in_ez_idle                  := "A-DBVALVES".ST6.STATION_MOVEMENT.test.IDLE_DUMMY
      );

      CALL "3STATE_DIAG"
      (  in_diag_status              := "A-DBVALVES".ST6.STATION_MOVEMENT.out.diag_status ,
         in_Ipw1                     := 'I170.2' ,
         in_Ipw2                     := ' ' ,
         in_Ipr1                     := 'I171.2' ,
         in_Ipr2                     := ' ' ,
         in_Qpw                      := 'Q170.6' ,
         in_Qpr                      := 'Q171.6' ,
         in_tio                      := "A-DBVALVES".io[32]
      );

      A "A-DBVALVES".ST6.STATION_MOVEMENT.out.alarm_hp;
      = "A-ALARMS".VALVES.err3.%X11;

      A "A-DBVALVES".ST6.STATION_MOVEMENT.out.alarm_wp;
      = "A-ALARMS".VALVES.err3.%X12;

      CALL "A-TESTSCL"
      (  in_nr                       := 32 ,
         out                         := "A-DBVALVES".ST6.STATION_MOVEMENT.test
      );

      A(;
      L "A-Doku_DB_OP".HMI.Manual_Functions;
      L 32;
      <>I;
      );
      R "A-DBVALVES".ST6.STATION_MOVEMENT.test.fp_HP;
      R "A-DBVALVES".ST6.STATION_MOVEMENT.test.fp_WP;
      R "A-DBVALVES".ST6.STATION_MOVEMENT.test.fp_IDLE;
NETWORK
TITLE = -

NETWORK
TITLE = [33] ST6 STACJA_MALY_SKOK - HP
//[33] ST6 STATION_SMALL_STEP - HP
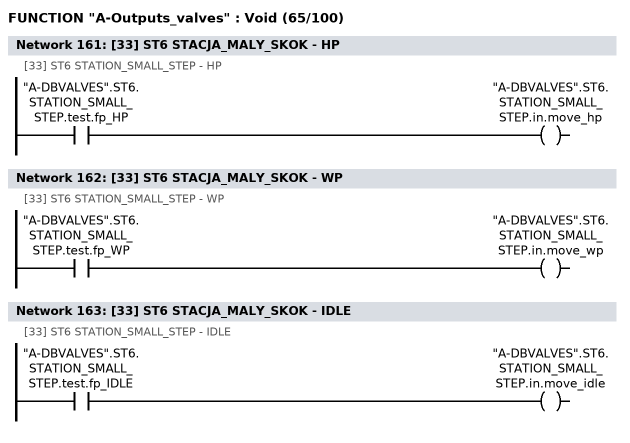
      O "A-DBVALVES".ST6.STATION_SMALL_STEP.test.fp_HP;
//    O     "A-Flags".STATION.IN_HP_STEP
      = "A-DBVALVES".ST6.STATION_SMALL_STEP.in.move_hp;
NETWORK
TITLE = [33] ST6 STACJA_MALY_SKOK - WP
//[33] ST6 STATION_SMALL_STEP - WP
      O "A-DBVALVES".ST6.STATION_SMALL_STEP.test.fp_WP;
      = "A-DBVALVES".ST6.STATION_SMALL_STEP.in.move_wp;
NETWORK
TITLE = [33] ST6 STACJA_MALY_SKOK - IDLE
//[33] ST6 STATION_SMALL_STEP - IDLE
      O "A-DBVALVES".ST6.STATION_SMALL_STEP.test.fp_IDLE;
      = "A-DBVALVES".ST6.STATION_SMALL_STEP.in.move_idle;
NETWORK
TITLE = [33] ST6 STACJA_MALY_SKOK
//[33] ST6 STATION_SMALL_STEP
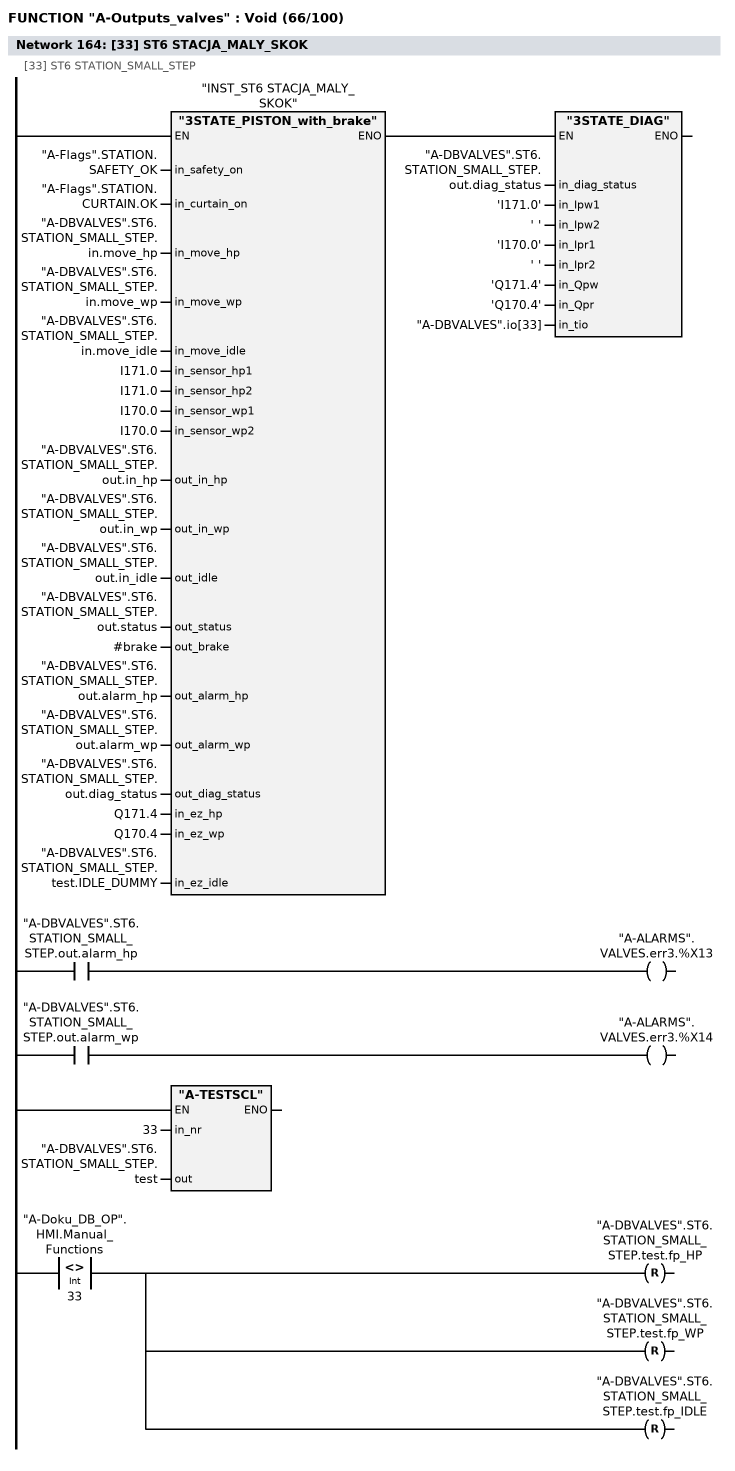
      CALL "3STATE_PISTON_with_brake", "INST_ST6 STACJA_MALY_SKOK"
      (  in_safety_on                := "A-Flags".STATION.SAFETY_OK ,
         in_curtain_on               := "A-Flags".STATION.CURTAIN.OK ,
         in_move_hp                  := "A-DBVALVES".ST6.STATION_SMALL_STEP.in.move_hp ,
         in_move_wp                  := "A-DBVALVES".ST6.STATION_SMALL_STEP.in.move_wp ,
         in_move_idle                := "A-DBVALVES".ST6.STATION_SMALL_STEP.in.move_idle ,
         in_sensor_hp1               := I171.0 ,
         in_sensor_hp2               := I171.0 ,
         in_sensor_wp1               := I170.0 ,
         in_sensor_wp2               := I170.0 ,
         out_in_hp                   := "A-DBVALVES".ST6.STATION_SMALL_STEP.out.in_hp ,
         out_in_wp                   := "A-DBVALVES".ST6.STATION_SMALL_STEP.out.in_wp ,
         out_idle                    := "A-DBVALVES".ST6.STATION_SMALL_STEP.out.in_idle ,
         out_status                  := "A-DBVALVES".ST6.STATION_SMALL_STEP.out.status ,
         out_brake                   := #brake ,
         out_alarm_hp                := "A-DBVALVES".ST6.STATION_SMALL_STEP.out.alarm_hp ,
         out_alarm_wp                := "A-DBVALVES".ST6.STATION_SMALL_STEP.out.alarm_wp ,
         out_diag_status             := "A-DBVALVES".ST6.STATION_SMALL_STEP.out.diag_status ,
         in_ez_hp                    := Q171.4 ,
         in_ez_wp                    := Q170.4 ,
         in_ez_idle                  := "A-DBVALVES".ST6.STATION_SMALL_STEP.test.IDLE_DUMMY
      );

      CALL "3STATE_DIAG"
      (  in_diag_status              := "A-DBVALVES".ST6.STATION_SMALL_STEP.out.diag_status ,
         in_Ipw1                     := 'I171.0' ,
         in_Ipw2                     := ' ' ,
         in_Ipr1                     := 'I170.0' ,
         in_Ipr2                     := ' ' ,
         in_Qpw                      := 'Q171.4' ,
         in_Qpr                      := 'Q170.4' ,
         in_tio                      := "A-DBVALVES".io[33]
      );

      A "A-DBVALVES".ST6.STATION_SMALL_STEP.out.alarm_hp;
      = "A-ALARMS".VALVES.err3.%X13;

      A "A-DBVALVES".ST6.STATION_SMALL_STEP.out.alarm_wp;
      = "A-ALARMS".VALVES.err3.%X14;

      CALL "A-TESTSCL"
      (  in_nr                       := 33 ,
         out                         := "A-DBVALVES".ST6.STATION_SMALL_STEP.test
      );

      A(;
      L "A-Doku_DB_OP".HMI.Manual_Functions;
      L 33;
      <>I;
      );
      R "A-DBVALVES".ST6.STATION_SMALL_STEP.test.fp_HP;
      R "A-DBVALVES".ST6.STATION_SMALL_STEP.test.fp_WP;
      R "A-DBVALVES".ST6.STATION_SMALL_STEP.test.fp_IDLE;
NETWORK
TITLE = -

NETWORK
TITLE = [34] ST6 STACJA_DUZY_SKOK - HP
//[34] ST6 STATION_BIG_STEP - HP
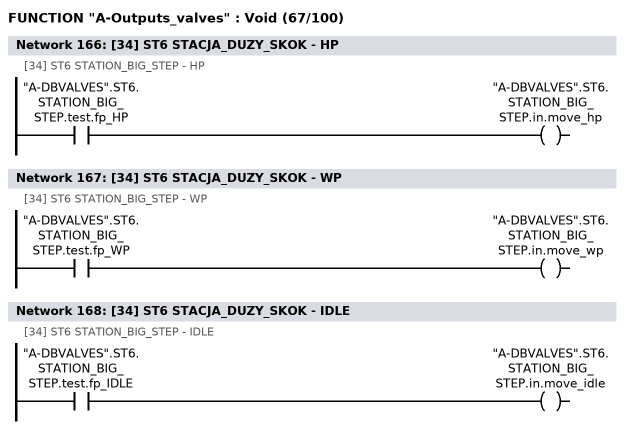
      O "A-DBVALVES".ST6.STATION_BIG_STEP.test.fp_HP;
//    O     "A-Flags".STATION.IN_HP_STEP
      = "A-DBVALVES".ST6.STATION_BIG_STEP.in.move_hp;
NETWORK
TITLE = [34] ST6 STACJA_DUZY_SKOK - WP
//[34] ST6 STATION_BIG_STEP - WP
      O "A-DBVALVES".ST6.STATION_BIG_STEP.test.fp_WP;
      = "A-DBVALVES".ST6.STATION_BIG_STEP.in.move_wp;
NETWORK
TITLE = [34] ST6 STACJA_DUZY_SKOK - IDLE
//[34] ST6 STATION_BIG_STEP - IDLE
      O "A-DBVALVES".ST6.STATION_BIG_STEP.test.fp_IDLE;
      = "A-DBVALVES".ST6.STATION_BIG_STEP.in.move_idle;
NETWORK
TITLE = [34] ST6 STACJA_DUZY_SKOK
//[34] ST6 STATION_BIG_STEP
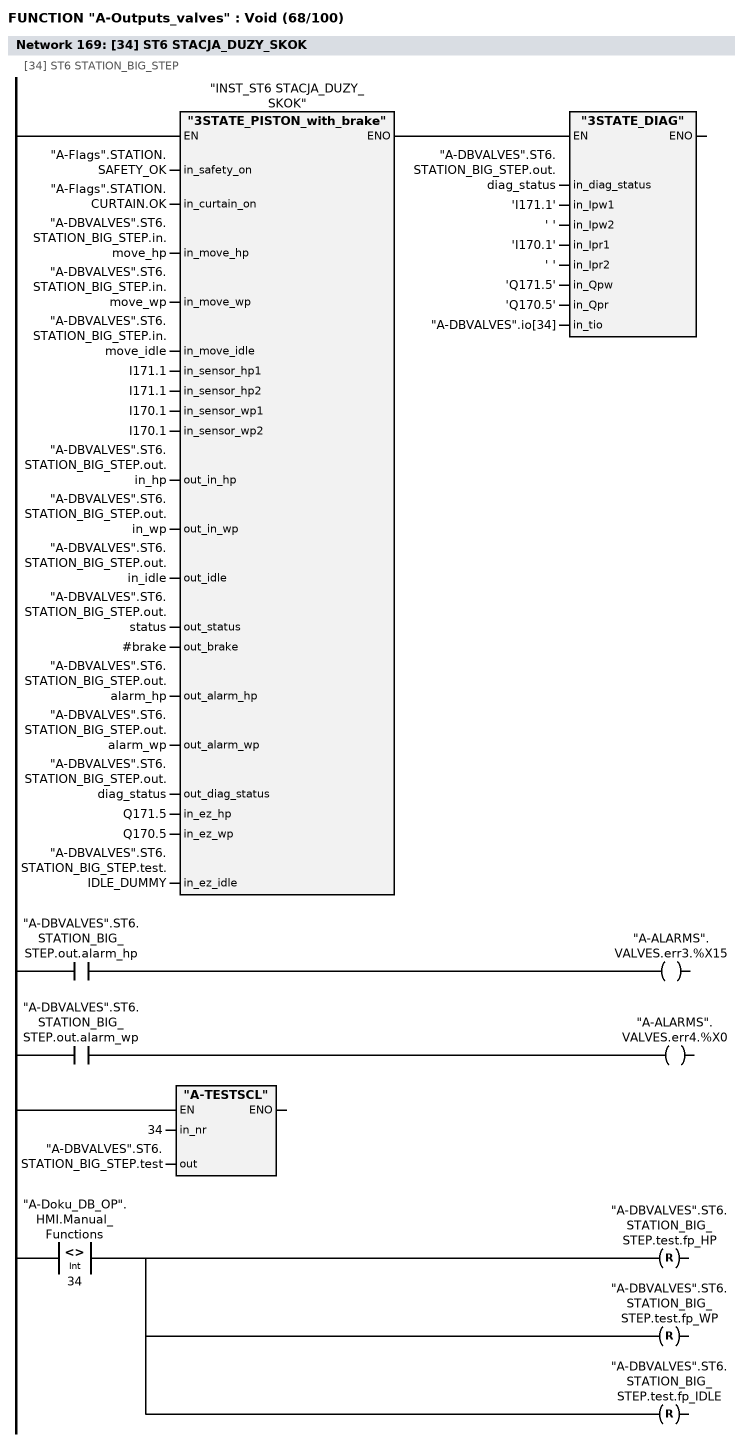
      CALL "3STATE_PISTON_with_brake", "INST_ST6 STACJA_DUZY_SKOK"
      (  in_safety_on                := "A-Flags".STATION.SAFETY_OK ,
         in_curtain_on               := "A-Flags".STATION.CURTAIN.OK ,
         in_move_hp                  := "A-DBVALVES".ST6.STATION_BIG_STEP.in.move_hp ,
         in_move_wp                  := "A-DBVALVES".ST6.STATION_BIG_STEP.in.move_wp ,
         in_move_idle                := "A-DBVALVES".ST6.STATION_BIG_STEP.in.move_idle ,
         in_sensor_hp1               := I171.1 ,
         in_sensor_hp2               := I171.1 ,
         in_sensor_wp1               := I170.1 ,
         in_sensor_wp2               := I170.1 ,
         out_in_hp                   := "A-DBVALVES".ST6.STATION_BIG_STEP.out.in_hp ,
         out_in_wp                   := "A-DBVALVES".ST6.STATION_BIG_STEP.out.in_wp ,
         out_idle                    := "A-DBVALVES".ST6.STATION_BIG_STEP.out.in_idle ,
         out_status                  := "A-DBVALVES".ST6.STATION_BIG_STEP.out.status ,
         out_brake                   := #brake ,
         out_alarm_hp                := "A-DBVALVES".ST6.STATION_BIG_STEP.out.alarm_hp ,
         out_alarm_wp                := "A-DBVALVES".ST6.STATION_BIG_STEP.out.alarm_wp ,
         out_diag_status             := "A-DBVALVES".ST6.STATION_BIG_STEP.out.diag_status ,
         in_ez_hp                    := Q171.5 ,
         in_ez_wp                    := Q170.5 ,
         in_ez_idle                  := "A-DBVALVES".ST6.STATION_BIG_STEP.test.IDLE_DUMMY
      );

      CALL "3STATE_DIAG"
      (  in_diag_status              := "A-DBVALVES".ST6.STATION_BIG_STEP.out.diag_status ,
         in_Ipw1                     := 'I171.1' ,
         in_Ipw2                     := ' ' ,
         in_Ipr1                     := 'I170.1' ,
         in_Ipr2                     := ' ' ,
         in_Qpw                      := 'Q171.5' ,
         in_Qpr                      := 'Q170.5' ,
         in_tio                      := "A-DBVALVES".io[34]
      );

      A "A-DBVALVES".ST6.STATION_BIG_STEP.out.alarm_hp;
      = "A-ALARMS".VALVES.err3.%X15;

      A "A-DBVALVES".ST6.STATION_BIG_STEP.out.alarm_wp;
      = "A-ALARMS".VALVES.err4.%X0;

      CALL "A-TESTSCL"
      (  in_nr                       := 34 ,
         out                         := "A-DBVALVES".ST6.STATION_BIG_STEP.test
      );

      A(;
      L "A-Doku_DB_OP".HMI.Manual_Functions;
      L 34;
      <>I;
      );
      R "A-DBVALVES".ST6.STATION_BIG_STEP.test.fp_HP;
      R "A-DBVALVES".ST6.STATION_BIG_STEP.test.fp_WP;
      R "A-DBVALVES".ST6.STATION_BIG_STEP.test.fp_IDLE;
NETWORK
TITLE = -

NETWORK
TITLE = [35] ST6 PIN - HP
//[35] ST6 PIN - HP
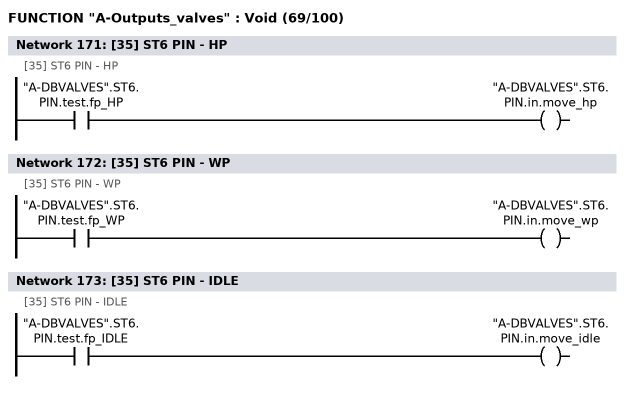
      O "A-DBVALVES".ST6.PIN.test.fp_HP;
//    O     "A-Flags".STATION.IN_HP_STEP
      = "A-DBVALVES".ST6.PIN.in.move_hp;
NETWORK
TITLE = [35] ST6 PIN - WP
//[35] ST6 PIN - WP
      O "A-DBVALVES".ST6.PIN.test.fp_WP;
      = "A-DBVALVES".ST6.PIN.in.move_wp;
NETWORK
TITLE = [35] ST6 PIN - IDLE
//[35] ST6 PIN - IDLE
      O "A-DBVALVES".ST6.PIN.test.fp_IDLE;
      = "A-DBVALVES".ST6.PIN.in.move_idle;
NETWORK
TITLE = [35] ST6 PIN
//[35] ST6 PIN
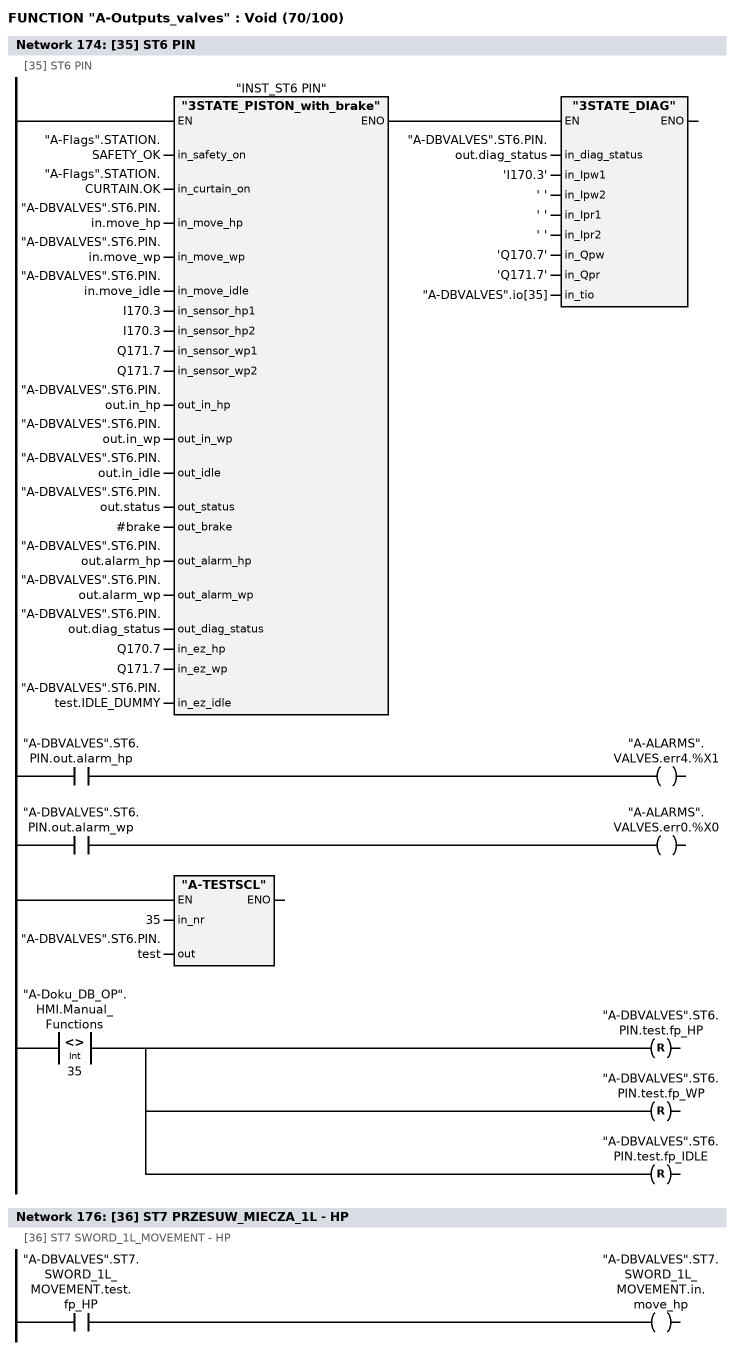
      CALL "3STATE_PISTON_with_brake", "INST_ST6 PIN"
      (  in_safety_on                := "A-Flags".STATION.SAFETY_OK ,
         in_curtain_on               := "A-Flags".STATION.CURTAIN.OK ,
         in_move_hp                  := "A-DBVALVES".ST6.PIN.in.move_hp ,
         in_move_wp                  := "A-DBVALVES".ST6.PIN.in.move_wp ,
         in_move_idle                := "A-DBVALVES".ST6.PIN.in.move_idle ,
         in_sensor_hp1               := I170.3 ,
         in_sensor_hp2               := I170.3 ,
         in_sensor_wp1               := Q171.7 ,
         in_sensor_wp2               := Q171.7 ,
         out_in_hp                   := "A-DBVALVES".ST6.PIN.out.in_hp ,
         out_in_wp                   := "A-DBVALVES".ST6.PIN.out.in_wp ,
         out_idle                    := "A-DBVALVES".ST6.PIN.out.in_idle ,
         out_status                  := "A-DBVALVES".ST6.PIN.out.status ,
         out_brake                   := #brake ,
         out_alarm_hp                := "A-DBVALVES".ST6.PIN.out.alarm_hp ,
         out_alarm_wp                := "A-DBVALVES".ST6.PIN.out.alarm_wp ,
         out_diag_status             := "A-DBVALVES".ST6.PIN.out.diag_status ,
         in_ez_hp                    := Q170.7 ,
         in_ez_wp                    := Q171.7 ,
         in_ez_idle                  := "A-DBVALVES".ST6.PIN.test.IDLE_DUMMY
      );

      CALL "3STATE_DIAG"
      (  in_diag_status              := "A-DBVALVES".ST6.PIN.out.diag_status ,
         in_Ipw1                     := 'I170.3' ,
         in_Ipw2                     := ' ' ,
         in_Ipr1                     := ' ' ,
         in_Ipr2                     := ' ' ,
         in_Qpw                      := 'Q170.7' ,
         in_Qpr                      := 'Q171.7' ,
         in_tio                      := "A-DBVALVES".io[35]
      );

      A "A-DBVALVES".ST6.PIN.out.alarm_hp;
      = "A-ALARMS".VALVES.err4.%X1;

      A "A-DBVALVES".ST6.PIN.out.alarm_wp;
      = "A-ALARMS".VALVES.err0.%X0;

      CALL "A-TESTSCL"
      (  in_nr                       := 35 ,
         out                         := "A-DBVALVES".ST6.PIN.test
      );

      A(;
      L "A-Doku_DB_OP".HMI.Manual_Functions;
      L 35;
      <>I;
      );
      R "A-DBVALVES".ST6.PIN.test.fp_HP;
      R "A-DBVALVES".ST6.PIN.test.fp_WP;
      R "A-DBVALVES".ST6.PIN.test.fp_IDLE;
NETWORK
TITLE = -

NETWORK
TITLE = [36] ST7 PRZESUW_MIECZA_1L - HP
//[36] ST7 SWORD_1L_MOVEMENT - HP
      O "A-DBVALVES".ST7.SWORD_1L_MOVEMENT.test.fp_HP;
//    O     "A-Flags".STATION.IN_HP_STEP
      = "A-DBVALVES".ST7.SWORD_1L_MOVEMENT.in.move_hp;
NETWORK
TITLE = [36] ST7 PRZESUW_MIECZA_1L - WP
//[36] ST7 SWORD_1L_MOVEMENT - WP
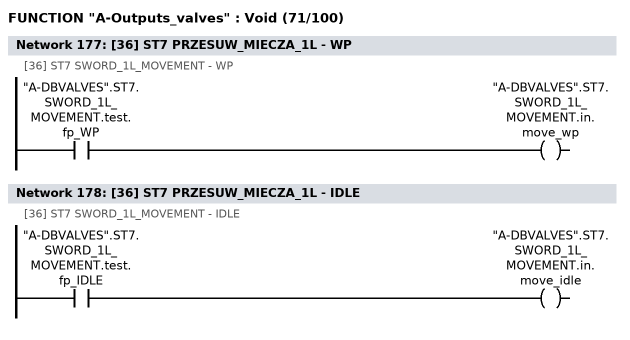
      O "A-DBVALVES".ST7.SWORD_1L_MOVEMENT.test.fp_WP;
      = "A-DBVALVES".ST7.SWORD_1L_MOVEMENT.in.move_wp;
NETWORK
TITLE = [36] ST7 PRZESUW_MIECZA_1L - IDLE
//[36] ST7 SWORD_1L_MOVEMENT - IDLE
      O "A-DBVALVES".ST7.SWORD_1L_MOVEMENT.test.fp_IDLE;
      = "A-DBVALVES".ST7.SWORD_1L_MOVEMENT.in.move_idle;
NETWORK
TITLE = [36] ST7 PRZESUW_MIECZA_1L
//[36] ST7 SWORD_1L_MOVEMENT
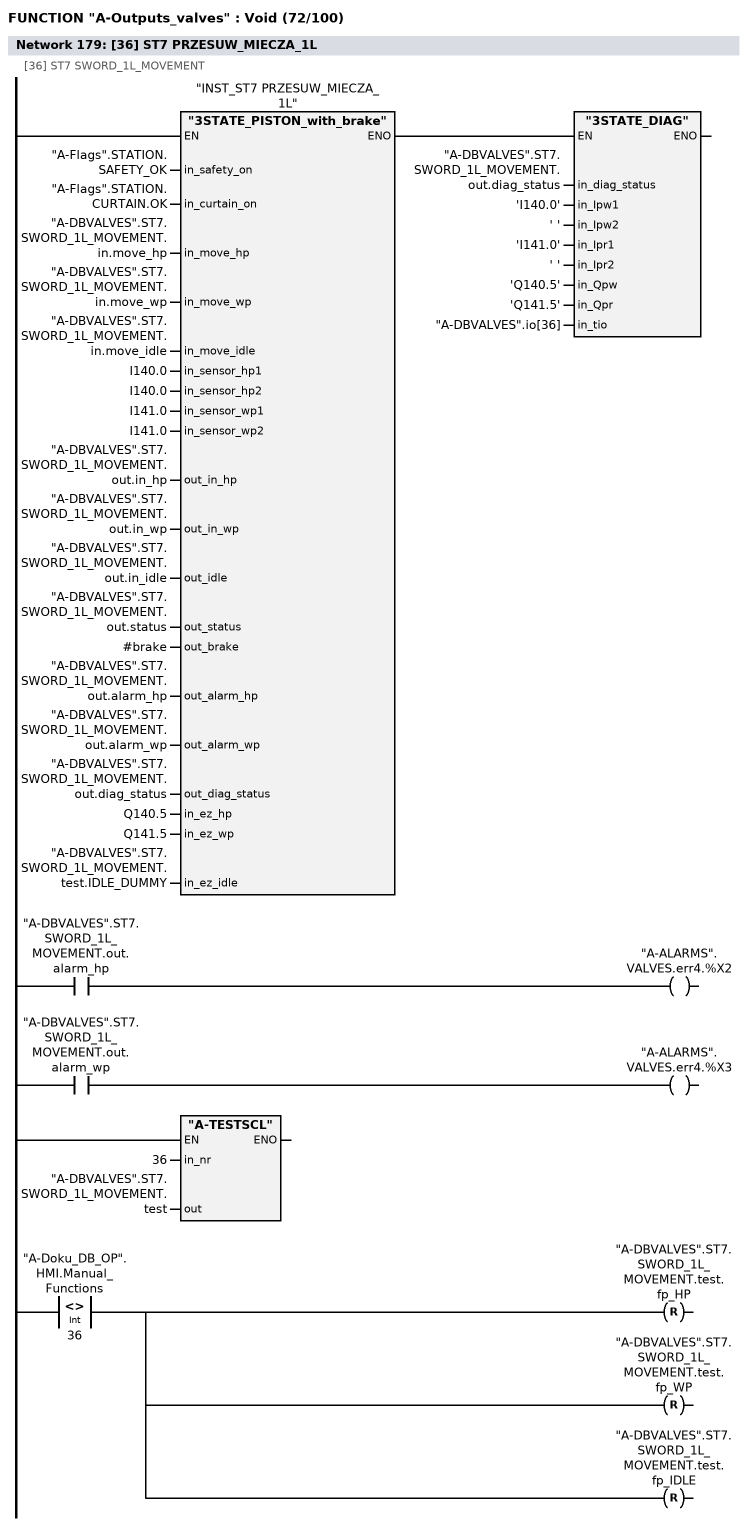
      CALL "3STATE_PISTON_with_brake", "INST_ST7 PRZESUW_MIECZA_1L"
      (  in_safety_on                := "A-Flags".STATION.SAFETY_OK ,
         in_curtain_on               := "A-Flags".STATION.CURTAIN.OK ,
         in_move_hp                  := "A-DBVALVES".ST7.SWORD_1L_MOVEMENT.in.move_hp ,
         in_move_wp                  := "A-DBVALVES".ST7.SWORD_1L_MOVEMENT.in.move_wp ,
         in_move_idle                := "A-DBVALVES".ST7.SWORD_1L_MOVEMENT.in.move_idle ,
         in_sensor_hp1               := I140.0 ,
         in_sensor_hp2               := I140.0 ,
         in_sensor_wp1               := I141.0 ,
         in_sensor_wp2               := I141.0 ,
         out_in_hp                   := "A-DBVALVES".ST7.SWORD_1L_MOVEMENT.out.in_hp ,
         out_in_wp                   := "A-DBVALVES".ST7.SWORD_1L_MOVEMENT.out.in_wp ,
         out_idle                    := "A-DBVALVES".ST7.SWORD_1L_MOVEMENT.out.in_idle ,
         out_status                  := "A-DBVALVES".ST7.SWORD_1L_MOVEMENT.out.status ,
         out_brake                   := #brake ,
         out_alarm_hp                := "A-DBVALVES".ST7.SWORD_1L_MOVEMENT.out.alarm_hp ,
         out_alarm_wp                := "A-DBVALVES".ST7.SWORD_1L_MOVEMENT.out.alarm_wp ,
         out_diag_status             := "A-DBVALVES".ST7.SWORD_1L_MOVEMENT.out.diag_status ,
         in_ez_hp                    := Q140.5 ,
         in_ez_wp                    := Q141.5 ,
         in_ez_idle                  := "A-DBVALVES".ST7.SWORD_1L_MOVEMENT.test.IDLE_DUMMY
      );

      CALL "3STATE_DIAG"
      (  in_diag_status              := "A-DBVALVES".ST7.SWORD_1L_MOVEMENT.out.diag_status ,
         in_Ipw1                     := 'I140.0' ,
         in_Ipw2                     := ' ' ,
         in_Ipr1                     := 'I141.0' ,
         in_Ipr2                     := ' ' ,
         in_Qpw                      := 'Q140.5' ,
         in_Qpr                      := 'Q141.5' ,
         in_tio                      := "A-DBVALVES".io[36]
      );

      A "A-DBVALVES".ST7.SWORD_1L_MOVEMENT.out.alarm_hp;
      = "A-ALARMS".VALVES.err4.%X2;

      A "A-DBVALVES".ST7.SWORD_1L_MOVEMENT.out.alarm_wp;
      = "A-ALARMS".VALVES.err4.%X3;

      CALL "A-TESTSCL"
      (  in_nr                       := 36 ,
         out                         := "A-DBVALVES".ST7.SWORD_1L_MOVEMENT.test
      );

      A(;
      L "A-Doku_DB_OP".HMI.Manual_Functions;
      L 36;
      <>I;
      );
      R "A-DBVALVES".ST7.SWORD_1L_MOVEMENT.test.fp_HP;
      R "A-DBVALVES".ST7.SWORD_1L_MOVEMENT.test.fp_WP;
      R "A-DBVALVES".ST7.SWORD_1L_MOVEMENT.test.fp_IDLE;
NETWORK
TITLE = -

NETWORK
TITLE = [37] ST7 PRZESUW_MIECZA_1P - HP
//[37] ST7 SWORD_1R_MOVEMENT - HP
